# EPICS substitutions: apps/jscalerApp/Db/jscalers_CTOF_FADC_sums.substitutions
file "db/jscalers_CTOF_FADC_sums.db" {
    pattern {SIDE}
    {"U"}
    {"D"}
}
